PROGRAM Sequence
VAR
	eState : E_State;
	
	ChargeRlyDelayON_Timer  : TON;
	ChargeRlyDelayDONE		: BOOL;
	ChargeRlyDelayON_PT		: TIME := T#250MS; //used for delay close and delay open for safe mode
	AbortPSnRlyDelay_Timer	: TON;
	AbortPSnRlyDelay_PT		: TIME := T#5MS; //defualt is 5ms
	AbortPSnRlyDelayDONE	: BOOL;
	ChargeCompleted			: BOOL;
	ChargingRunOutTMR_TON	: TON;
	ChargingRunOutTMR_ET	: TIME;
	ChargedRunOutTMR_TON	: TON;
	ChargedRunOutTMR_ET		: TIME;
	FireToSafeDelayTMR_TON	: TON;
	FireToSafeDelayTMR_PT	: TIME := T#5S;
	FireToSafeDelayTMR_ET	: TIME;
	FirePBpressed			: BOOL := FALSE;
	ShotFired				: BOOL := FALSE;
	
	ShotTrigDelayTMR_TON	: LTON;
	ShotTrigDelayTMR_PT		: LTIME := LTIME#10US;
	ShotTrigDelayTMR_ET		: LTIME;
	
	ShotTrigPulseTMR_TON	: LTON;
	ShotTrigPulseTMR_PT		: LTIME := LTIME#1S + ShotTrigDelayTMR_PT;
	ShotTrigPulseTMR_ET		: LTIME;
		
	ScopeTrigPulseTMR_TON	: TON;
	ScopeTrigPulseTMR_PT	: TIME := T#10MS;
	ScopeTrigPulseTMR_ET	: TIME;
	
	DumpingRunOutTMR_TON 	: TON;
	DumpingRunOutTMR_PT		: TIME := T#10S;
	DumpingRunOutTMR_ET		: TIME;
	LocalDumpActive			: BOOL := FALSE;

	StartChargingBroadcast	: BOOL := FALSE;
	StartCharger			: ARRAY[1..7] OF BOOL;

	ChargeTimeFinished		: BOOL;
	StartCharWarningTMR_TON : TON;
	StartCharWarningTMR_PT	: TIME := T#0S;  //no need to warning
	StartCharWarningTMR_ET	: TIME;
	ChargeDelayStart		: BOOL := FALSE;
	
	DumpRlyDelayTMR_TON		: TON;
	DumpRlyDelay_PT			: TIME := T#250MS;
	DumpRlyDelay_ET			: TIME;
	
	i						: INT := 1; //1-7 chargers
	j						: INT := 1; //1-8 Shaft ramp dump rly
	k						: INT := 1; //1-9
	m						: INT := 1; //4-6
	n 						: INT := 6;
	CompDumpStagger			: Stagger_FB;
	SRDumpStagger			: Stagger_FB;
END_VAR

//Critical Delay Time


//hv output delay
HMI_DB.HVONdelayPT := INT_TO_TIME (HMI_DB.HVONdelayPT_INT);
ChargeRlyDelayON_PT := HMI_DB.HVONdelayPT;

//runout timer
HMI_DB.RunOutTMR_PT := DINT_TO_TIME (HMI_DB.RunOutTMR_PT_INT*1000);
HMI_DB.RunOutTMR_elapse := (TIME_TO_DINT (HMI_DB.RunOutTMR_PT - ChargedRunOutTMR_TON.ET))/1000;
HMI_DB.ChargingRunOutTMR_elapse := TIME_TO_INT(ChargingRunOutTMR_TON.PT/1000 - ChargingRunOutTMR_TON.ET/1000);

//charge realy timer 
ChargeRlyDelayON_Timer(PT := ChargeRlyDelayON_PT);

//reset timer
IF eState <> E_State.CHARGING THEN 
	ChargingRunOutTMR_TON (IN := FALSE);
	//LCP1_IO.Segment[1].Module[1].ModuleCharged := FALSE; //for status light only

	FOR i := 1 TO n BY 1 DO
		ChargeTime_DB.ChargerDelay_TON[i] (IN := FALSE, PT := ChargeTime_DB.ChargerDelay_PT[i], ET => ChargeTime_DB.ChargerDelay_ET[i]);
		ChargeTime_DB.ChargingTimeElapse_TON[i].IN := FALSE;
		ChargeRlyDelayON_Timer (IN := FALSE);
	END_FOR;
	
END_IF

IF eState <> E_State.CHARGECOMPLETE THEN 
	//LCP1_IO.Segment[1].Module[1].ModuleCharged := FALSE; //for status light only
	ChargedRunOutTMR_TON (IN := FALSE); // only needed in charge complete
END_IF

IF HMI_DB.HMI_ManualModeSelected = TRUE AND eState = E_State.SAFE (*AND ChargeDelayStart = FALSE *)THEN //added charge delay start
	eState := E_State.ManualMode;
END_IF

IF eState = E_State.CHARGING OR eState = E_State.CHARGECOMPLETE OR eState = E_State.ABORT (*OR ChargeDelayStart = TRUE*) THEN //added charge delay start
	HMI_DB.HMI_ManualModeSelected := FALSE;
END_IF

IF eState <> E_State.ManualMode THEN
	HMI_DB.CloseChargeRlySW := FALSE;
	HMI_DB.OpenDumpRlySW := FALSE;
	HMI_DB.TurnChrgHVonSW := FALSE;
	HMI_DB.TurnChrgInhibitOffSW := FALSE;
	HMI_DB.TurnOnShotTrigSW := FALSE;
	HMI_DB.TurnOnChargeAlarm := FALSE;
END_IF

IF HMI_DB.DumpPB = TRUE OR plc_plc_comm_DB.ReadStateFromPLC = E_State.DUMPING THEN  //although will bring the state out of abort, it will go back to abort if faults are not clear.
	eState := E_State.DUMPING;
	ELSIF (HMI_DB.AbortPB = TRUE OR Trips_DB.TimerRunOutON = TRUE OR plc_plc_comm_DB.ReadStateFromPLC = E_State.ABORT) AND eState <> E_State.ManualMode THEN 
		eState := E_State.ABORT;
	//	ELSE
	//		eState := E_State.SAFE;
		END_IF;
		

CASE eState OF 
	//Safe OR IDLE
	E_State.SAFE:
		ChargeCompleted := FALSE;
		FirePBpressed := FALSE;
		FireToSafeDelayTMR_TON (IN := FALSE);
		ChargeRlyDelayON_Timer(IN:= FALSE);
		ChargeTime_DB.LongestChargeTime_TON (IN := FALSE); //reset timer
		ChargeTimeFinished := FALSE; //reset chargetime done bit
		ShotTrigDelayTMR_TON (IN := FALSE, PT := ShotTrigDelayTMR_PT, ET => ShotTrigDelayTMR_ET);
		ScopeTrigPulseTMR_TON (IN := FALSE, PT := ScopeTrigPulseTMR_PT, ET => ScopeTrigPulseTMR_ET);
		ShotTrigPulseTMR_TON (IN := FALSE, PT := ShotTrigPulseTMR_PT, ET => ShotTrigPulseTMR_ET);
		
		plc_plc_comm_DB.WriteStatetoPLC := E_state.SAFE;
		//MCP_IO.Fire := FALSE; //turn off all firing triggers
		
		
		(*	// might not have interlock	
		IF Permissives_DB.CageInterlockOK = TRUE AND HMI_DB.ArmTheCagePB = TRUE THEN 
			MCP_IO.EnergizeACKontactor := TRUE;
		END_IF;
		*)
		
		//TURN OFF ALL CHARGERS
		FOR i := 1 TO n BY 1 DO 
			MCP_IO.Charger[i].inhibit := TRUE; // inhibit = high, no output | inhibit = low, allows output
			
			//MCP_IO.Charger[i].voltageSP := 0.001;
			StartCharger[i] := FALSE; // reset bit
			ChargeTimeFinished := FALSE;
			StartChargingBroadcast := FALSE;
			//reset charger delay timer
			ChargeTime_DB.ChargerDelay_TON[i] (IN := FALSE, PT := ChargeTime_DB.ChargerDelay_PT[i], ET => ChargeTime_DB.ChargerDelay_ET[i]);
			ChargeTime_DB.ChargingTimeElapse_TON[i] (IN := FALSE); 
		END_FOR;
		ChargingRunOutTMR_TON (IN := FALSE);
		ChargedRunOutTMR_TON (IN := FALSE);
		DumpingRunOutTMR_TON (IN := FALSE);
		
		ScopeTrigPulseTMR_TON (IN := FALSE);
		ShotTrigDelayTMR_TON (IN := FALSE);
		ShotTrigPulseTMR_TON (IN := FALSE);
	
		MCP_IO.MagDriver[1].CloseChargeRly := FALSE;
		MCP_IO.MagDriver[2].CloseChargeRly := FALSE;
		MCP_IO.MagDriver[3].CloseChargeRly := FALSE;
		MCP_IO.MagDriver[4].CloseChargeRly := FALSE;
		MCP_IO.MagDriver[5].CloseChargeRly := FALSE;
		MCP_IO.MagDriver[6].CloseChargeRly := FALSE;
 
		//reset stagger fg
		CompDumpStagger (start := FALSE, n := 6, reset := TRUE); 

		FOR j := 1 TO 6 BY 1 DO 
			MCP_IO.MagDriver[j].OpenDumpRly := FALSE;
		END_FOR;
		
		IF HMI_DB.ChargePB = TRUE (*AND MCP_IO.EnergizeACKontactor*) OR plc_plc_comm_DB.ReadStateFromPLC = E_State.CHARGING THEN //directly sent from LV 
			ChargeDelayStart := TRUE;
		ELSIF HMI_DB.DumpPB = TRUE THEN
				eState := E_State.DUMPING; 
		END_IF;
		
		IF ChargeDelayStart = TRUE AND Permissives_DB.AllDumpResTempOK = TRUE THEN //if dump resistors are too hot, it won't go to charge
			// turn on warning light  
			MCP_IO.TurnONSystemChargedLED := TRUE;
			//LCP2_IO.SegmentCharged := TRUE;
			//LCP3_IO.SegmentCharged := TRUE;
			StartCharWarningTMR_TON (IN := TRUE, PT := StartCharWarningTMR_PT, ET=> StartCharWarningTMR_ET);  //warning time is set to 0
		END_IF;
		
		IF StartCharWarningTMR_TON.Q = TRUE THEN 
			ChargeDelayStart := FALSE;
			StartCharWarningTMR_TON (IN := FALSE);
			eState := E_State.CHARGING;
		END_IF

	E_State.CHARGING:
		StartCharWarningTMR_TON (IN := FALSE, PT := StartCharWarningTMR_PT, ET=> StartCharWarningTMR_ET);
		ChargeDelayStart := FALSE;
		// turn on warning light  
		MCP_IO.TurnONSystemChargedLED := TRUE;
		
		FirePBpressed := FALSE;
		MCP_IO.TriggerSCRs := FALSE;
		
		plc_plc_comm_DB.WriteStatetoPLC := E_state.CHARGING;
		
		//start charging runout timer
		MCP_IO.MagDriver[1].CloseChargeRly := TRUE;
		MCP_IO.MagDriver[2].CloseChargeRly := TRUE;
		MCP_IO.MagDriver[3].CloseChargeRly := TRUE;
		MCP_IO.MagDriver[4].CloseChargeRly := TRUE;
		MCP_IO.MagDriver[5].CloseChargeRly := TRUE;
		MCP_IO.MagDriver[6].CloseChargeRly := TRUE;
	
		
		//stagger the relays - change the name later
		CompDumpStagger (start := TRUE, n := 6, reset := FALSE);
		//or make sure the turn reset on when turning off the dump relay outputs
		MCP_IO.MagDriver[1].OpenDumpRly := CompDumpStagger.OutputHi[1]; //turn output ON
		MCP_IO.MagDriver[2].OpenDumpRly := CompDumpStagger.OutputHi[2];
		MCP_IO.MagDriver[3].OpenDumpRly := CompDumpStagger.OutputHi[3];
		MCP_IO.MagDriver[4].OpenDumpRly := CompDumpStagger.OutputHi[4];
		MCP_IO.MagDriver[5].OpenDumpRly := CompDumpStagger.OutputHi[5];
		MCP_IO.MagDriver[6].OpenDumpRly := CompDumpStagger.OutputHi[6];
		
		IF CompDumpStagger.OutputHi[6] = TRUE THEN 
			CompDumpStagger.start := FALSE;
		END_IF
		
		//permissives to charge
		IF Permissives_DB.ReadyToCharge = TRUE THEN 
			FOR i := 1 TO n BY 1 DO 
				//MCP_IO.Charger[i].voltageSP := (HMI_DB.TDKLoad[i].RequiredChargedV *1000);
				MCP_IO.Charger[i].voltageSP := (HMI_DB.HPT5[i].RequiredChargedV);
			END_FOR
		END_IF
		
		//start charging runout timer
		ChargingRunOutTMR_TON (IN := TRUE, PT := (ChargeTime_DB.LongestChargeTime_PT + HMI_DB.RunOutTMR_PT), ET => ChargingRunOutTMR_ET);
		
		IF Trips_DB.ChargingTimerRunout = TRUE THEN 
			StartChargingBroadcast := FALSE; // reset the broadcast bit whne all chargers
			ChargeTimeFinished := FALSE; //reset chargetime done bit
			ChargingRunOutTMR_TON (IN := FALSE);
			FOR i := 1 TO n BY 1 DO 
				ChargeTime_DB.ChargingTimeElapse_TON[i] (IN := FALSE);							
			END_FOR
			
			eState := E_State.ABORT; 
		END_IF
		
		IF Permissives_DB.AllChargeRelayClosed = TRUE THEN
			//start broadcasting on charger timer
			StartChargingBroadcast := TRUE;
		END_IF;
		// ******might not have a charge time stagger... all just go on at once ******
		//start timer 
		IF StartChargingBroadcast = TRUE THEN 
			//start total charge time TIMER
			ChargeTime_DB.LongestChargeTime_TON (IN := TRUE, PT := ChargeTime_DB.LongestChargeTime_PT, ET => ChargeTime_DB.LongestChargeTime_ET);
			
			//mapping HMI Charger Voltage SP to MCP IO 
			FOR i := 1 TO n BY 1 DO
				MCP_IO.Charger[i].voltageSP := (HMI_DB.HPT5[i].RequiredChargedV );
				//MCP_IO.Charger[1].voltageSP := REAL_TO_DINT (Setpoints.TDKLoad[1].RequiredChargedV);
			END_FOR;
			
			// delay stagger starts here
			ChargeTime_DB.ChargerDelay_TON[1] (IN := TRUE, PT := ChargeTime_DB.ChargerDelay_PT[1], ET => ChargeTime_DB.ChargerDelay_ET[1]);
			ChargeTime_DB.ChargerDelay_TON[2] (IN := TRUE, PT := ChargeTime_DB.ChargerDelay_PT[2], ET => ChargeTime_DB.ChargerDelay_ET[2]);
			ChargeTime_DB.ChargerDelay_TON[3] (IN := TRUE, PT := ChargeTime_DB.ChargerDelay_PT[3], ET => ChargeTime_DB.ChargerDelay_ET[3]);
		
			ChargeTime_DB.ChargerDelay_TON[4] (IN := TRUE, PT := ChargeTime_DB.ChargerDelay_PT[4], ET => ChargeTime_DB.ChargerDelay_ET[4]);
			ChargeTime_DB.ChargerDelay_TON[5] (IN := TRUE, PT := ChargeTime_DB.ChargerDelay_PT[5], ET => ChargeTime_DB.ChargerDelay_ET[5]);
			ChargeTime_DB.ChargerDelay_TON[6] (IN := TRUE, PT := ChargeTime_DB.ChargerDelay_PT[6], ET => ChargeTime_DB.ChargerDelay_ET[6]);
			
			ELSE
				//Turn inhibit High on all chargers and all timer if no broadcasting
				FOR i := 1 TO n BY 1 DO 
					MCP_IO.Charger[i].inhibit := TRUE; 
					// turn off timer
					ChargeTime_DB.ChargerDelay_TON[i] (IN := FALSE, PT := ChargeTime_DB.ChargerDelay_PT[i], ET => ChargeTime_DB.ChargerDelay_ET[i]);
				END_FOR;
		END_IF;
			
		FOR i := 1 TO n BY 1 DO	
			//turn on HV output to load	
			IF ChargeTime_DB.ChargerDelay_TON[i].Q = TRUE THEN
				StartCharger[i] := TRUE;
			END_IF	
			
			IF StartCharger[i] = TRUE (*AND Permissives.ReadyToCharge = TRUE*) THEN
				MCP_IO.Charger[i].inhibit := FALSE;
				ChargeTime_DB.ChargerDelay_TON[i] (IN := FALSE, PT := ChargeTime_DB.ChargerDelay_PT[i], ET => ChargeTime_DB.ChargerDelay_ET[i]);
				ChargeTime_DB.ChargingTimeElapse_TON[i]  (IN := TRUE, PT := REAL_TO_TIME (1000*MCP_IO.Charger[i].ChargeTime.timeToChargeLoad));
				//cal 
			END_IF;
			
			IF ChargeTime_DB.ChargingTimeElapse_TON[i].Q THEN
				StartCharger[i] := FALSE;
				ChargeTime_DB.ChargingTimeElapse_TON[i] (IN := FALSE); 
				//ChargeTime_DB.ChargerDelay_TON[i] (IN := FALSE, PT := ChargeTime_DB.ChargerDelay_PT[i], ET => ChargeTime_DB.ChargerDelay_ET[i]);
			END_IF;
		END_FOR;
				
		IF ChargingRunOutTMR_TON.Q = TRUE THEN
			Trips_DB.ChargingTimerRunout := TRUE;
			ChargingRunOutTMR_TON (IN := FALSE);
		END_IF;
		
		IF ChargeTime_DB.LongestChargeTime_TON.Q = TRUE THEN 
			ChargeTimeFinished := TRUE;
			StartChargingBroadcast := FALSE;
		
			ChargeTime_DB.LongestChargeTime_TON (IN := FALSE); //reset timer
		END_IF
		
		IF ChargeTimeFinished = TRUE THEN 
			
			FOR i := 1 TO n BY 1 DO 
				StartCharger[i] := FALSE;
				ChargeTime_DB.ChargingTimeElapse_TON[i] (IN := FALSE);							
			END_FOR
		END_IF
		
		//condition for charge complete
		IF (Permissives_DB.AllChargerEOC = TRUE AND 
			ChargeTimeFinished = TRUE (*all voltage reached*)) OR plc_plc_comm_DB.ReadStateFromPLC = E_State.CHARGECOMPLETE  
			THEN 
				ChargeCompleted := TRUE;
		//ELSE
			//ChargeCompleted := FALSE;
		END_IF
		
//if cap voltage feedback >= charger setpoints && EOC && all timer runout then chargecomplete
		IF ChargeCompleted = TRUE THEN 
			FOR i := 1 TO n BY 1 DO 
				
				MCP_IO.Charger[i].inhibit := TRUE;
				
				StartCharger[i] := FALSE;
				ChargeTime_DB.ChargingTimeElapse_TON[i] (IN := FALSE);	
			END_FOR;
			ChargeRlyDelayON_Timer ( IN := TRUE, PT := ChargeRlyDelayON_PT);
		END_IF;

		IF ChargeRlyDelayON_Timer.Q = TRUE THEN
			ChargeRlyDelayDONE := TRUE;
		END_IF;

		IF ChargeRlyDelayDONE = TRUE THEN 	
			//Open all relays
			MCP_IO.MagDriver[1].CloseChargeRly := FALSE;
			MCP_IO.MagDriver[2].CloseChargeRly := FALSE;
			MCP_IO.MagDriver[3].CloseChargeRly := FALSE;	
			MCP_IO.MagDriver[4].CloseChargeRly := FALSE;
			MCP_IO.MagDriver[5].CloseChargeRly := FALSE;
			MCP_IO.MagDriver[6].CloseChargeRly := FALSE;	
				
		//stagger the output - probably don't need to recheck this
//			LCP1_IO.Segment[1].OpenModule1To3DumpRly := TRUE;
//			LCP1_IO.Segment[2].OpenModule4To6DumpRly := TRUE;
//			LCP1_IO.Segment[3].OpenModule7To9DumpRly := TRUE;
//			LCP2_IO.Segment[4].OpenModule1To3DumpRly := TRUE;
//			LCP2_IO.Segment[5].OpenModule4To6DumpRly := TRUE;
//			LCP2_IO.Segment[6].OpenModule7To9DumpRly := TRUE;
			//shaft ramp - also does not need to recheck
			
			ChargeRlyDelayON_Timer ( IN := FALSE, PT := ChargeRlyDelayON_PT);							
			StartChargingBroadcast := FALSE; // reset the broadcast bit whne all chargers 
			
			eState := E_State.CHARGECOMPLETE;
		END_IF
		
	
	E_State.CHARGECOMPLETE:
		//keep led light on
		MCP_IO.TurnONSystemChargedLED := TRUE;
		
		ChargeRlyDelayDONE := FALSE;
		ChargeCompleted := FALSE;
		StartChargingBroadcast := FALSE; // reset the broadcast bit whne all chargers 
		ChargedRunOutTMR_TON (IN := TRUE, PT := HMI_DB.RunOutTMR_PT);
		ChargeRlyDelayON_Timer ( IN := FALSE, PT := ChargeRlyDelayON_PT);
		
		plc_plc_comm_DB.WriteStatetoPLC := E_state.CHARGECOMPLETE; //status to M1 PP
		
		IF HMI_DB.FirePB = TRUE OR plc_plc_comm_DB.Button.FirePBPressed = TRUE THEN 
			//LCP1_IO.Segment[1].Module[1].Fire := TRUE;
			MCP_IO.TriggerScope := TRUE;
			
			ChargedRunOutTMR_TON (IN := FALSE);
			//and all other shot triggers.
			FirePBpressed := TRUE;
			//ELSE
				//LCP1_IO.Segment[1].Module[1].Fire := FALSE;
		END_IF
		
		IF FirePBpressed = TRUE THEN 
			//FireToSafeDelayTMR_TON (IN := TRUE, PT := FireToSafeDelayTMR_PT, ET => FireToSafeDelayTMR_ET);
			ShotTrigDelayTMR_TON (IN := TRUE, PT := ShotTrigDelayTMR_PT, ET => ShotTrigDelayTMR_ET);
			ScopeTrigPulseTMR_TON (IN := TRUE, PT := ScopeTrigPulseTMR_PT, ET => ScopeTrigPulseTMR_ET);
			ShotTrigPulseTMR_TON (IN := TRUE, PT := ShotTrigPulseTMR_PT, ET => ShotTrigPulseTMR_ET);
			//LCP1_IO.Segment[1].Module[1].Fire := TRUE;
		END_IF
		
		IF ScopeTrigPulseTMR_TON.Q = TRUE THEN 
			MCP_IO.TriggerScope := FALSE;
			
			//ScopeTrigPulseTMR_TON (IN := FALSE);
		END_IF
		
		IF ShotTrigDelayTMR_TON.Q = TRUE THEN
			MCP_IO.TriggerSCRs := TRUE;
			
			ShotFired := TRUE;
			//ShotTrigDelayTMR_TON (IN := FALSE);
		END_IF
		//might need to be a nested elsif
		IF ShotTrigPulseTMR_TON.Q = TRUE THEN
			MCP_IO.TriggerSCRs := FALSE;
			
			//ShotTrigPulseTMR_TON (IN := FALSE);
		END_IF
		
		IF ShotFired = TRUE THEN
			FireToSafeDelayTMR_TON (IN := TRUE, PT := FireToSafeDelayTMR_PT, ET => FireToSafeDelayTMR_ET);
		END_IF
		
		IF FireToSafeDelayTMR_TON.Q = TRUE THEN
			FirePBpressed := FALSE;
			ShotFired := FALSE;
			FireToSafeDelayTMR_TON (IN := FALSE);
			ScopeTrigPulseTMR_TON (IN := FALSE);
			ShotTrigDelayTMR_TON (IN := FALSE);
			ShotTrigPulseTMR_TON (IN := FALSE);
			//LCP1_IO.Segment[1].Module[1].TriggerScope := FALSE;
			eState := E_State.SAFE;
		END_IF;
		
		IF ChargedRunOutTMR_TON.Q = TRUE THEN
			Trips_DB.ChargedTimerRunout := TRUE;
			ChargeTimeFinished := FALSE; //reset chargetime done bit
			ChargedRunOutTMR_TON (IN := FALSE);
			ScopeTrigPulseTMR_TON (IN := FALSE);
			ShotTrigDelayTMR_TON (IN := FALSE);
			ShotTrigPulseTMR_TON (IN := FALSE);
			eState := E_State.ABORT;
		END_IF

	E_State.DUMPING:

		// dump all 
		CompDumpStagger (start := FALSE, n := 6, reset := TRUE);
		MCP_IO.MagDriver[1].OpenDumpRly := FALSE;
		MCP_IO.MagDriver[2].OpenDumpRly := FALSE;
		MCP_IO.MagDriver[3].OpenDumpRly := FALSE;
		MCP_IO.MagDriver[4].OpenDumpRly := FALSE;
		MCP_IO.MagDriver[5].OpenDumpRly := FALSE;
		MCP_IO.MagDriver[6].OpenDumpRly := FALSE;
		
		FOR i := 1 TO n BY 1 DO 
			MCP_IO.Charger[i].voltageSP := 0.001;
			MCP_IO.Charger[i].inhibit := TRUE;
		END_FOR;
		
		MCP_IO.MagDriver[1].CloseChargeRly := FALSE;
		MCP_IO.MagDriver[2].CloseChargeRly := FALSE;
		MCP_IO.MagDriver[3].CloseChargeRly := FALSE;
		
		MCP_IO.MagDriver[4].CloseChargeRly := FALSE;
		MCP_IO.MagDriver[5].CloseChargeRly := FALSE;
		MCP_IO.MagDriver[6].CloseChargeRly := FALSE;
		
		ChargeDelayStart := FALSE;
		FirePBpressed := FALSE;
		StartCharWarningTMR_TON (IN := FALSE, PT := StartCharWarningTMR_PT, ET=> StartCharWarningTMR_ET);
				
		DumpingRunOutTMR_TON (IN := TRUE, PT := DumpingRunOutTMR_PT);
		
		plc_plc_comm_DB.WriteStatetoPLC := E_state.DUMPING; //status to M1 PP
		
		//HMI_DB.CloseChargeRlySW := FALSE;
		//HMI_DB.OpenDumpRlySW := FALSE;
		
		IF DumpingRunOutTMR_TON.Q = TRUE AND Permissives_DB.AllCapsDischarged = TRUE THEN
			eState := E_State.SAFE;
		END_IF

	E_State.ABORT:
		//dump all
		FOR i := 1 TO n BY 1 DO
			MCP_IO.Charger[i].inhibit := TRUE;
			
			MCP_IO.Charger[i].voltageSP := 0.001;
		END_FOR
				
		MCP_IO.MagDriver[1].CloseChargeRly := FALSE;
		MCP_IO.MagDriver[2].CloseChargeRly := FALSE;
		MCP_IO.MagDriver[3].CloseChargeRly := FALSE;
		
		MCP_IO.MagDriver[4].CloseChargeRly := FALSE;
		MCP_IO.MagDriver[5].CloseChargeRly := FALSE;
		MCP_IO.MagDriver[6].CloseChargeRly := FALSE;
		
		//reset stagger fg 
		CompDumpStagger (start := FALSE, n := 6, reset := TRUE);
		MCP_IO.MagDriver[1].OpenDumpRly := FALSE;
		MCP_IO.MagDriver[2].OpenDumpRly := FALSE;
		MCP_IO.MagDriver[3].OpenDumpRly := FALSE;
		MCP_IO.MagDriver[4].OpenDumpRly := FALSE;
		MCP_IO.MagDriver[5].OpenDumpRly := FALSE;
		MCP_IO.MagDriver[6].OpenDumpRly := FALSE;
		
		HMI_DB.CloseChargeRlySW := FALSE;
		HMI_DB.OpenDumpRlySW := FALSE;
		HMI_DB.TurnChrgHVonSW := FALSE;
		HMI_DB.TurnChrgInhibitOffSW := FALSE;
		HMI_DB.TurnOnShotTrigSW := FALSE;
		HMI_DB.TurnOnChargeAlarm := FALSE;
		
		MCP_IO.TriggerSCRs := FALSE;
		
		
		StartCharWarningTMR_TON (IN := FALSE);
		ChargeDelayStart := FALSE;
		FirePBpressed := FALSE;
		
		plc_plc_comm_DB.WriteStatetoPLC := E_state.ABORT; //status to M1 PP
	
		IF Permissives_DB.SystemIsSafe = TRUE AND Trips_DB.TimerRunOutON = FALSE THEN
			eState := E_State.SAFE;
		END_IF
		
	E_State.ManualMode:
		
		plc_plc_comm_DB.WriteStatetoPLC := E_state.ManualMode; //status to M1 PP
		
		DumpingRunOutTMR_TON (IN := FALSE);
		StartCharWarningTMR_TON (IN := FALSE); // note
		
		MCP_IO.MagDriver[1].CloseChargeRly := MCP_IO.MagDriver[2].CloseChargeRly := MCP_IO.MagDriver[3].CloseChargeRly := HMI_DB.CloseChargeRlySW;
		MCP_IO.MagDriver[4].CloseChargeRly := MCP_IO.MagDriver[5].CloseChargeRly := MCP_IO.MagDriver[6].CloseChargeRly := HMI_DB.CloseChargeRlySW;
		
		MCP_IO.MagDriver[1].OpenDumpRly := MCP_IO.MagDriver[2].OpenDumpRly := MCP_IO.MagDriver[3].OpenDumpRly := HMI_DB.OpenDumpRlySW;
		MCP_IO.MagDriver[4].OpenDumpRly := MCP_IO.MagDriver[5].OpenDumpRly := MCP_IO.MagDriver[6].OpenDumpRly := HMI_DB.OpenDumpRlySW;
		
	
		IF HMI_DB.TurnChrgInhibitOffSW = TRUE THEN 
			FOR i := 1 TO n BY 1 DO 
				MCP_IO.Charger[i].inhibit := FALSE;
			END_FOR
			ELSE
				FOR i := 1 TO n BY 1 DO 
					MCP_IO.Charger[i].inhibit := TRUE;
				END_FOR				
		END_IF
		
		MCP_IO.TriggerSCRs := HMI_DB.TurnOnShotTrigSW;
		MCP_IO.TurnONSystemChargedLED := HMI_DB.TurnOnChargeAlarm;
		
		IF HMI_DB.HMI_ManualModeSelected = FALSE THEN
			eState := E_State.SAFE;
		END_IF
		
END_CASE;

IF i > n THEN 
	i := 1;
END_IF;	

IF j > 6 THEN 
	j := 1;
END_IF;	

IF k > 9 THEN 
	k := 1;
END_IF;	

IF m > 6 THEN 
	m := 4;
END_IF;

END_PROGRAM

(* stored: Version 1.1.0.1, ProductVersion 3.1.4024.11
   POU Sequence: Id {3c03c824-1ca6-44f0-8304-54f7bd72a17b}, SpecialFunc None *)
